FUNCTION_BLOCK ReqPanelLift_HMI (* Service Interface Function Block Type *)
  (* Standard: 61499-2 *)
  (* Version 0.0, 6/3/2016, Andrei, nxtControl GmbH, template *)
  PACKAGE Main;
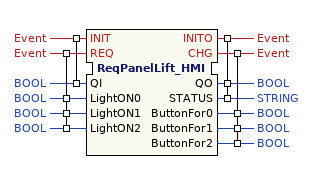
  EVENT_INPUT
    INIT WITH QI;
    REQ WITH LightON0, LightON1, LightON2;
  END_EVENT
  EVENT_OUTPUT
    INITO WITH QO, STATUS;
    CHG WITH ButtonFor0, ButtonFor1, ButtonFor2;
  END_EVENT
  VAR_INPUT
    QI : BOOL;
    LightON0 : BOOL;
    LightON1 : BOOL;
    LightON2 : BOOL;
  END_VAR
  VAR_OUTPUT
    QO : BOOL; (* Event Output Qualifier *)
    STATUS : STRING; (* Service Status *)
    ButtonFor0 : BOOL;
    ButtonFor1 : BOOL;
    ButtonFor2 : BOOL;
  END_VAR
END_FUNCTION_BLOCK
